FUNCTION_BLOCK ModbusReadWordArray EXTENDS ModbusIo
VAR_INPUT
END_VAR
VAR_OUTPUT
	Value: ARRAY [1..125] OF WORD;
	Text: string;
END_VAR
VAR
END_VAR
VAR PERSISTENT
END_VAR

SUPER^();
Text := GetText();

METHOD GetText : string
VAR_INPUT
END_VAR
VAR
	Str: STRING;
	arr: ARRAY [1..125] OF WORD;
	p: POINTER TO ARRAY [0..MAX_STRING_LENGTH] OF BYTE;
	n: int;
	{attribute 'TcEncoding':='UTF-8'}
	Utf8: STRING;
END_VAR
arr := Value;
FOR n := 1 TO 125 DO
	arr[n] := SHR(arr[n] AND 16#FF00, 8) + SHL(arr[n] AND 16#00FF, 8);
END_FOR
p := ADR(arr);
Str := BYTEARR_TO_MAXSTRING(p^);
STRING_TO_UTF8(ADR(Utf8), ADR(Str), SIZEOF(Utf8));
GetText := Utf8;
END_METHOD

PROPERTY ValueWordArray : array [1..125] of WORD
GET
ValueWordArray := Value;
END_GET
SET
Value := ValueWordArray;
END_SET
END_PROPERTY

END_FUNCTION_BLOCK

(* stored: Version 1.1.0.1, ProductVersion 3.1.4024.6
   POU ModbusReadWordArray: Id {d68fbbc9-ad32-4387-b6cd-bb784ee837ef}, SpecialFunc None
   Method GetText: Id {ffea3707-997a-43f6-91b6-15d08933b010}
   Property ValueWordArray: Id {839f9df0-1a28-460e-baa6-1a213d09aaf8}
   Get Get: Id {b74c2e47-683a-4ea7-8526-163b11e96bde}
   Set Set: Id {ecd8b270-fe8a-4589-9a6f-9a1e0abc5946} *)
